INTERFACE ITF_CAMover

METHOD AddMoverToThisGroup : HRESULT
VAR_INPUT
	MoverToAdd : ITF_XtsMoverAxis;
END_VAR
END_METHOD

METHOD RemoveAMover : BOOL
VAR_INPUT
	moverId : UDINT;
END_VAR
END_METHOD

END_INTERFACE

(* stored: Version 1.1.0.1
   Itf ITF_CAMover: Id {7d0eb89e-eb46-4416-8384-7e72bbf5d44b}
   Method AddMoverToThisGroup: Id {b77778eb-2994-4a80-ac40-69283ff8c14c}
   Method RemoveAMover: Id {d4388b6a-db0d-4c22-9a5b-3ffbb622a3ca} *)
